FUNCTION_BLOCK PICKER_MODEL_TYPE1_TEST (* Composite Function Block Type *)
  (* Standard: 61499-2 *)
  (* Version 0.2, 2003-12-05, JHC, Rockwell Automation, Renamed from NEWCOMPFB. *)
  (* Version 0.1, 2002-01-08, JHC, Rockwell Automation, Added DLY FB as example. *)
  (* Version 0.0, 2000-05-27, JHC, Rockwell Automation *)
  (* Compiler header: package fb.rt.pnp; *)
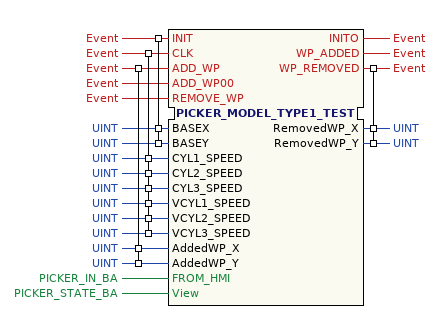
  EVENT_INPUT
    INIT WITH BASEX, BASEY; (* Initialisation *)
    CLK WITH CYL1_SPEED, CYL2_SPEED, CYL3_SPEED, VCYL1_SPEED, VCYL2_SPEED, VCYL3_SPEED;
    ADD_WP WITH AddedWP_X, AddedWP_Y;
    ADD_WP00;
    REMOVE_WP;
  END_EVENT
  EVENT_OUTPUT
    INITO; (* Initialization Confirm *)
    WP_ADDED;
    WP_REMOVED WITH RemovedWP_X, RemovedWP_Y;
  END_EVENT
  VAR_INPUT
    BASEX : UINT;
    BASEY : UINT;
    CYL1_SPEED : UINT;
    CYL2_SPEED : UINT;
    CYL3_SPEED : UINT;
    VCYL1_SPEED : UINT;
    VCYL2_SPEED : UINT;
    VCYL3_SPEED : UINT;
    AddedWP_X : UINT;
    AddedWP_Y : UINT;
  END_VAR
  VAR_OUTPUT
    RemovedWP_X : UINT;
    RemovedWP_Y : UINT;
  END_VAR
  SOCKETS
    FROM_HMI : PICKER_IN_BA;
    View : PICKER_STATE_BA;
  END_SOCKETS
  FBS
    Model : ModelBA;
    Control : MasterSlave_TEST;
  END_FBS
  EVENT_CONNECTIONS
    INIT TO Model.INIT;
    Model.INITO TO View.INIT;
    CLK TO Model.CLK;
    ADD_WP TO Model.ADD_WP;
    REMOVE_WP TO Model.REMOVE_WP;
    Model.WP_ADDED TO WP_ADDED;
    Model.WP_REMOVED TO WP_REMOVED;
    ADD_WP00 TO Model.ADD_WP00;
    Model.CNF TO View.CHG;
    FROM_HMI.REQ TO Model.REQ;
    Model.INITO TO Control.INIT;
    Model.CHG TO Control.REQ;
    Control.INITO TO INITO;
    Control.CNF TO Model.CYL_IND;
    CLK TO Control.REQ;
  END_CONNECTIONS
  DATA_CONNECTIONS
    Model.BASE_X TO View.BASE_X;
    Model.BASE_Y TO View.BASE_Y;
    Model.CYL1_X TO View.CYL1_X;
    Model.CYL1_Y TO View.CYL1_Y;
    Model.CYL2_X TO View.CYL2_X;
    Model.CYL2_Y TO View.CYL2_Y;
    Model.VCYL1_X TO View.VCYL1_X;
    Model.VCYL1_Y TO View.VCYL1_Y;
    Model.WP1_X TO View.WP1_X;
    Model.WP1_Y TO View.WP1_Y;
    Model.VACUUM_ON TO View.VACUUM_ON;
    BASEX TO Model.BASEX;
    BASEY TO Model.BASEY;
    CYL1_SPEED TO Model.CYL1_SPEED;
    CYL2_SPEED TO Model.CYL2_SPEED;
    VCYL1_SPEED TO Model.VCYL1_SPEED;
    AddedWP_X TO Model.AddedWP_X;
    AddedWP_Y TO Model.AddedWP_Y;
    Model.RemovedWP_X TO RemovedWP_X;
    Model.RemovedWP_Y TO RemovedWP_Y;
    Model.WP3_X TO View.WP3_X;
    Model.WP3_Y TO View.WP3_Y;
    Model.WP2_X TO View.WP2_X;
    Model.WP2_Y TO View.WP2_Y;
    FROM_HMI.add1 TO Model.Add1;
    FROM_HMI.add2 TO Model.Add2;
    FROM_HMI.add3 TO Model.Add3;
    Model.VACUUM_ON TO Control.vacuum;
    Model.pp0 TO Control.pp0;
    Model.pp1 TO Control.pp1;
    Model.pp2 TO Control.pp2;
    Model.pp3 TO Control.pp3;
    Model.CYL3_Y TO View.CYL3_Y;
    Model.CYL3_X TO View.CYL3_X;
    Model.VCYL2_X TO View.VCYL2_X;
    Model.VCYL2_Y TO View.VCYL2_Y;
    Model.VCYL3_X TO View.VCYL3_X;
    Model.VCYL3_Y TO View.VCYL3_Y;
    Model.WP4_X TO View.WP4_X;
    Model.WP4_Y TO View.WP4_Y;
    FROM_HMI.add4 TO Model.Add4;
    CYL3_SPEED TO Model.CYL3_SPEED;
    VCYL2_SPEED TO Model.VCYL2_SPEED;
    VCYL3_SPEED TO Model.VCYL3_SPEED;
    Model.cyl1home TO Control.cyl1home;
    Model.cyl1end TO Control.cyl1end;
    Model.cyl2home TO Control.cyl2home;
    Model.cyl2end TO Control.cyl2end;
    Model.cyl3home TO Control.cyl3home;
    Model.cyl3end TO Control.cyl3end;
    Model.vcyl1home TO Control.vcyl1home;
    Model.vcyl1end TO Control.vcyl1end;
    Model.vcyl2home TO Control.vcyl2home;
    Model.vcyl2end TO Control.vcyl2end;
    Model.vcyl3home TO Control.vcyl3home;
    Model.vcyl3end TO Control.vcyl3end;
    Model.pp4 TO Control.pp4;
    Control.venturi_on TO Model.vacuum_on;
    Control.venturi_off TO Model.vacuum_off;
    Control.cyl1MoveOut TO Model.cyl1_fwd;
    Control.cyl2MoveOut TO Model.cyl2_fwd;
    Control.cyl3MoveOut TO Model.cyl3_fwd;
    Control.cyl3MoveIn TO Model.cyl3_back;
    Control.vcyl1MoveOut TO Model.vcyl1_down;
    Control.vcyl2MoveOut TO Model.vcyl2_down;
    Control.vcyl3MoveOut TO Model.vcyl3_down;
    Model.cyl3mid TO Control.cyl3mid;
  END_CONNECTIONS
END_FUNCTION_BLOCK
